PROGRAM Alias
VAR
	i : INT := 1; //mag driver index
	n : INT := 6; //mag driver num
	j : INT := 1; //1-2
	m : INT := 2; //# of ultra cap per driver rack
	k : INT := 1; //ultra cap number 
	
	p : INT := 12; //# of ultra caps = 12
END_VAR

//R1 : MCP**  
	//INPUT
	//AI - EL3068
	MCP_IO.MagDriver[1].ShotCurrentFeedback_raw	:= Input.R1_01_00; //
	MCP_IO.MagDriver[2].ShotCurrentFeedback_raw	:= Input.R1_01_01; //
	MCP_IO.MagDriver[3].ShotCurrentFeedback_raw	:= Input.R1_01_02; // 
	MCP_IO.MagDriver[4].ShotCurrentFeedback_raw	:= Input.R1_01_03; //
	MCP_IO.MagDriver[5].ShotCurrentFeedback_raw	:= Input.R1_01_04; // 
	MCP_IO.MagDriver[6].ShotCurrentFeedback_raw	:= Input.R1_01_05; //  
	//Spare										:= Input.R1_01_06; //  
	//Spare										:= Input.R1_01_07; //
	
	//DI
	MCP_IO.MagDriver[1].DumpResistorTemp_raw	:= Input.R1_02_00; //
	MCP_IO.MagDriver[2].DumpResistorTemp_raw	:= Input.R1_02_01; // 
	MCP_IO.MagDriver[3].DumpResistorTemp_raw	:= Input.R1_02_02; // 
	MCP_IO.MagDriver[4].DumpResistorTemp_raw	:= Input.R1_02_03; // 
	MCP_IO.MagDriver[5].DumpResistorTemp_raw	:= Input.R1_02_04; // 
	MCP_IO.MagDriver[6].DumpResistorTemp_raw	:= Input.R1_02_05; // 
	
	MCP_IO.MagDriver[1].SCR_ready_to_fire		:= Input.R1_03_00; // 
	MCP_IO.MagDriver[2].SCR_ready_to_fire		:= Input.R1_03_01; // 
	MCP_IO.MagDriver[3].SCR_ready_to_fire		:= Input.R1_03_02; // 
	MCP_IO.MagDriver[4].SCR_ready_to_fire		:= Input.R1_03_03; // 
	MCP_IO.MagDriver[5].SCR_ready_to_fire		:= Input.R1_03_04; // 
	MCP_IO.MagDriver[6].SCR_ready_to_fire		:= Input.R1_03_05; // 
	
	MCP_IO.MagDriver[1].ChargeRelayClose		:= Input.R1_04_00; //
	MCP_IO.MagDriver[2].ChargeRelayClose		:= Input.R1_04_01; //
	MCP_IO.MagDriver[3].ChargeRelayClose		:= Input.R1_04_02; //
	MCP_IO.MagDriver[4].ChargeRelayClose		:= Input.R1_04_03; //
	MCP_IO.MagDriver[5].ChargeRelayClose		:= Input.R1_04_04; //
	MCP_IO.MagDriver[6].ChargeRelayClose		:= Input.R1_04_05; //
	
	//DQ
	Output.R1_05_00	:= MCP_IO.MagDriver[1].CloseChargeRly;
	Output.R1_05_01	:= MCP_IO.MagDriver[2].CloseChargeRly;
	Output.R1_05_02	:= MCP_IO.MagDriver[3].CloseChargeRly;
	Output.R1_05_03	:= MCP_IO.MagDriver[4].CloseChargeRly;
	Output.R1_05_04	:= MCP_IO.MagDriver[5].CloseChargeRly;
	Output.R1_05_05	:= MCP_IO.MagDriver[6].CloseChargeRly;
	//Output.R1_05_06	:= 
	//Output.R1_05_07	:= 
	
	//DQ
	Output.R1_06_00	:= MCP_IO.MagDriver[1].OpenDumpRly;
	Output.R1_06_01	:= MCP_IO.MagDriver[2].OpenDumpRly;
	Output.R1_06_02	:= MCP_IO.MagDriver[3].OpenDumpRly;
	Output.R1_06_03	:= MCP_IO.MagDriver[4].OpenDumpRly;
	Output.R1_06_04 := MCP_IO.MagDriver[5].OpenDumpRly;
	Output.R1_06_05 := MCP_IO.MagDriver[6].OpenDumpRly;
	Output.R1_06_06 := MCP_IO.TriggerScope;
	
	MCP_IO.MagDriver[1].DumpRelayOpen		:= Input.R1_07_00; //
	MCP_IO.MagDriver[2].DumpRelayOpen		:= Input.R1_07_01; //
	MCP_IO.MagDriver[3].DumpRelayOpen		:= Input.R1_07_02; //
	MCP_IO.MagDriver[4].DumpRelayOpen		:= Input.R1_07_03; //
	MCP_IO.MagDriver[5].DumpRelayOpen		:= Input.R1_07_04; //
	MCP_IO.MagDriver[6].DumpRelayOpen		:= Input.R1_07_05; //
	(*shaft ramp add below*)
	
	//DQ
	Output.R1_08_00	:= MCP_IO.Charger[1].inhibit;
	Output.R1_08_01	:= MCP_IO.Charger[2].inhibit;
	Output.R1_08_02	:= MCP_IO.Charger[3].inhibit;
	Output.R1_08_03	:= MCP_IO.Charger[4].inhibit;
	Output.R1_08_04	:= MCP_IO.Charger[5].inhibit;
	Output.R1_08_05	:= MCP_IO.Charger[6].inhibit;
	Output.R1_08_06 := MCP_IO.TriggerSCRs;
	Output.R1_08_07	:= MCP_IO.TurnONSystemChargedLED;
		
	//EL4008 AQ
	Output.R1_09_00	:= MCP_IO.Charger[1].voltageSP_raw;
	Output.R1_09_01	:= MCP_IO.Charger[2].voltageSP_raw;
	Output.R1_09_02	:= MCP_IO.Charger[3].voltageSP_raw;
	Output.R1_09_03	:= MCP_IO.Charger[4].voltageSP_raw;	
	Output.R1_09_04	:= MCP_IO.Charger[5].voltageSP_raw;
	Output.R1_09_05	:= MCP_IO.Charger[6].voltageSP_raw;
	
	//CANBUS 
	//Output.R1_10_CANrequest := CAN_comm.
	Output.R1_10_CANrequest.cobId := MCP_IO.MagDriver[1].Cap[1].CanTx_config_ID;
	Output.R1_10_CANrequest.data[0] := MCP_IO.MagDriver[1].Cap[1].CanTx_config_request[0];
	Output.R1_10_CANrequest.data[1] := MCP_IO.MagDriver[1].Cap[1].CanTx_config_request[1];
	Output.R1_10_CANrequest.data[2] := MCP_IO.MagDriver[1].Cap[1].CanTx_config_request[2];
	Output.R1_10_CANrequest.data[3] := MCP_IO.MagDriver[1].Cap[1].CanTx_config_request[3];
	Output.R1_10_CANrequest.data[4] := MCP_IO.MagDriver[1].Cap[1].CanTx_config_request[4];
	Output.R1_10_CANrequest.data[5] := MCP_IO.MagDriver[1].Cap[1].CanTx_config_request[5];
	Output.R1_10_CANrequest.data[6] := MCP_IO.MagDriver[1].Cap[1].CanTx_config_request[6];
	Output.R1_10_CANrequest.data[7] := MCP_IO.MagDriver[1].Cap[1].CanTx_config_request[7];
	
	// P1 PP comm
	HMI_DB.ClearFaultPB := plc_plc_comm_DB.Button.ClearAllFaults;
	HMI_DB.FirePB 		:= plc_plc_comm_DB.Button.FirePBPressed;
	HMI_DB.DumpPB 		:= plc_plc_comm_DB.Button.DumpPB;

	//MCP_IO.MagDriver[1].Cap[1].Elec_AveVolt 		:= Input.R1_10_CapNumber[1].Status.Elec_AveVolt; //per cell <- example
	//this is replaced by the loop below
(*	MCP_IO.MagDriver[1].Cap[1].Elec_AveVolt 		:= Input.R1_10_CapNumber[1].Status.Elec_AveVolt; //per cell
	MCP_IO.MagDriver[1].Cap[1].Elec_Balancing 		:= Input.R1_10_CapNumber[1].Status.Elec_Balancing; // 0x0[Not Active], 0x1[Active], 0x2[Error], 0x3[Not Available]
	MCP_IO.MagDriver[1].Cap[1].Elec_HighestVolt 	:= Input.R1_10_CapNumber[1].Status.Elec_HighestVolt; //per cell
	MCP_IO.MagDriver[1].Cap[1].Elec_Imbalance 		:= Input.R1_10_CapNumber[1].Status.Elec_Imbalance;  // 0x0[No Warnings], 0x1[Warning Active], 0x2[Alarm Active], 0x3[Not Available]
	MCP_IO.MagDriver[1].Cap[1].Elec_OverVoltage		:= Input.R1_10_CapNumber[1].Status.Elec_OverVoltage;  // 0x0[No Warnings], 0x1[Warning Active], 0x2[Alarm Active], 0x3[NOT Available] 
	MCP_IO.MagDriver[1].Cap[1].Elec_VoltageSum		:= Input.R1_10_CapNumber[1].Status.Elec_VoltageSum; //total voltage in one UC
	MCP_IO.MagDriver[1].Cap[1].Therm_HighestCell	:= Input.R1_10_CapNumber[1].Status.Therm_HighestCell; //C
	MCP_IO.MagDriver[1].Cap[1].Therm_HighTemp		:= Input.R1_10_CapNumber[1].Status.Therm_HighTemp;  //0x0[No Warnings], 0x1[Warning Active], 0x2[Alarm Active], 0x3[NOT Available]
*)	
//need to verify the couunter
	FOR i := 1 TO n BY 1 DO 
		FOR j := 1 TO m BY 1 DO 
			IF j = 1 THEN 
				k := 2*i -j;
				ELSIF j = 2 THEN 
					k :=j*i;
			END_IF

			MCP_IO.MagDriver[i].Cap[j].Elec_AveVolt			:= Input.R1_10_CapNumber[k].Elec_AveVolt; //per cell
			MCP_IO.MagDriver[i].Cap[j].Elec_Balancing		:= Input.R1_10_CapNumber[k].Elec_Balancing; // 0x0[Not Active], 0x1[Active], 0x2[Error], 0x3[Not Available]
			MCP_IO.MagDriver[i].Cap[j].Elec_HighestVolt		:= Input.R1_10_CapNumber[k].Elec_HighestVolt; //per cell
			MCP_IO.MagDriver[i].Cap[j].Elec_Imbalance		:= Input.R1_10_CapNumber[k].Elec_Imbalance;  // 0x0[No Warnings], 0x1[Warning Active], 0x2[Alarm Active], 0x3[Not Available]
			MCP_IO.MagDriver[i].Cap[j].Elec_OverVoltage		:= Input.R1_10_CapNumber[k].Elec_OverVoltage;  // 0x0[No Warnings], 0x1[Warning Active], 0x2[Alarm Active], 0x3[NOT Available] 
			MCP_IO.MagDriver[i].Cap[j].Elec_VoltageSum		:= Input.R1_10_CapNumber[k].Elec_VoltageSum; //total voltage in one UC
			MCP_IO.MagDriver[i].Cap[j].Therm_HighestCell	:= Input.R1_10_CapNumber[k].Therm_HighestCell; //C
			MCP_IO.MagDriver[i].Cap[j].Therm_HighTemp		:= Input.R1_10_CapNumber[k].Therm_HighTemp;  //0x0[No Warnings], 0x1[Warning Active], 0x2[Alarm Active], 0x3[NOT Available]

		END_FOR		
	END_FOR
	
	MCP_IO.MagDriver[1].Cap[1].UltraCap_Dummy.R1_10_UC_Rx_cobID := Input.R1_10_UC_7F_status.R1_10_UC_Rx_cobID;
	MCP_IO.MagDriver[1].Cap[1].UltraCap_Dummy.R1_10_UC_Rx_data := Input.R1_10_UC_7F_status.R1_10_UC_Rx_data;	
	// need to have how many voltage monitor board or voltage transmitter board per fruit stand ????
	//LCP3_IO.VMB.VTB[1].

	//LV Alias
	//commented out to test the sequence
	(*
	HMI_DB.ChargePB 				:= LV.TxWord1.0;
	HMI_DB.DumpPB					:= LV.TxWord1.1;		
	HMI_DB.AbortPB					:= LV.TxWord1.2;
	HMI_DB.FirePB					:= LV.TxWord1.3;
	HMI_DB.ClearFaultPB 			:= LV.TxWord1.4;
	HMI_DB.AllDumpRelaysOpenBP		:= LV.TxWord1.5;
	HMI_DB.AllChargeRelayCloseBP	:= LV.TxWord1.6;
	HMI_DB.SystemSafeBP				:= LV.TxWord1.7;
	HMI_DB.CloseChargeRlySW			:= LV.TxWord1.8;
	HMI_DB.OpenDumpRlySW 			:= LV.TxWord1.9;
	HMI_DB.HMI_ManualModeSelected	:= LV.TxWord1.10;  // 1 = manual mode selected
	HMI_DB.TurnChrgHVonSW			:= LV.TxWord1.11;
	HMI_DB.TurnChrgInhibitOffSW		:= LV.TxWord1.12;
	HMI_DB.TurnOnShotTrigSW			:= LV.TxWord1.13;
	HMI_DB.TurnOnChargeAlarm		:= LV.TxWord1.14;
	HMI_DB.AllVoltMonBoardStatusOKBP:= LV.TxWord1.15;
	//not sure if you want to control these via LV
	(*
	MCP_IO.Charger[1].HV_ON			:= LV.TxWord2.0;
	MCP_IO.Charger[1].inhibit		:= LV.TxWord2.1;
	MCP_IO.Charger[2].HV_ON			:= LV.TxWord2.2;
	MCP_IO.Charger[2].inhibit		:= LV.TxWord2.3;
	
	MCP_IO.Charger[3].HV_ON			:= LV.TxWord2.4;
	MCP_IO.Charger[3].inhibit		:= LV.TxWord2.5;
	MCP_IO.Charger[4].HV_ON			:= LV.TxWord2.6;
	MCP_IO.Charger[4].inhibit		:= LV.TxWord2.7;
	MCP_IO.Charger[5].HV_ON			:= LV.TxWord2.8;
	MCP_IO.Charger[5].inhibit		:= LV.TxWord2.9;
	MCP_IO.Charger[6].HV_ON			:= LV.TxWord2.10;
	MCP_IO.Charger[6].inhibit		:= LV.TxWord2.11;
	HMI_DB.HMI_DB.AllDumpRelaysCloseBP := LV.TxWord2.12;
	*)
	
	LV.RxWord1.0 := LV.Charger[1].EndOfCharge			:= MCP_IO.Charger[1].EndOfCharge;
	LV.RxWord1.1 := LV.Charger[1].HV_isON				:= MCP_IO.Charger[1].HV_isON;
	LV.RxWord1.2 := LV.Charger[1].inhibited				:= MCP_IO.Charger[1].inhibited;
	LV.RxWord1.3 := LV.Charger[1].SummaryFaulted		:= MCP_IO.Charger[1].SummaryFaulted;
	LV.RxWord1.4 := LV.Charger[2].EndOfCharge			:= MCP_IO.Charger[2].EndOfCharge;
	LV.RxWord1.5 := LV.Charger[2].HV_isON				:= MCP_IO.Charger[2].HV_isON;
	LV.RxWord1.6 := LV.Charger[2].inhibited				:= MCP_IO.Charger[2].inhibited;
	LV.RxWord1.7 := LV.Charger[2].SummaryFaulted		:= MCP_IO.Charger[2].SummaryFaulted;
	LV.RxWord1.8 := LV.Charger[3].EndOfCharge			:= MCP_IO.Charger[3].EndOfCharge;
	LV.RxWord1.9 := LV.Charger[3].HV_isON				:= MCP_IO.Charger[3].HV_isON;
	LV.RxWord1.10 := LV.Charger[3].inhibited			:= MCP_IO.Charger[3].inhibited;
	LV.RxWord1.11 := LV.Charger[3].SummaryFaulted		:= MCP_IO.Charger[3].SummaryFaulted;
	LV.RxWord1.12 := LV.Charger[4].EndOfCharge			:= MCP_IO.Charger[4].EndOfCharge;
	LV.RxWord1.13 := LV.Charger[4].HV_isON				:= MCP_IO.Charger[4].HV_isON;
	LV.RxWord1.14 := LV.Charger[4].inhibited			:= MCP_IO.Charger[4].inhibited;
	LV.RxWord1.15 := LV.Charger[4].SummaryFaulted		:= MCP_IO.Charger[4].SummaryFaulted;
	
	LV.RxWord2.0 := LV.Charger[5].EndOfCharge			:= MCP_IO.Charger[5].EndOfCharge;
	LV.RxWord2.1 := LV.Charger[5].HV_isON				:= MCP_IO.Charger[5].HV_isON;
	LV.RxWord2.2 := LV.Charger[5].inhibited				:= MCP_IO.Charger[5].inhibited;
	LV.RxWord2.3 := LV.Charger[5].SummaryFaulted		:= MCP_IO.Charger[5].SummaryFaulted;
	LV.RxWord2.4 := LV.Charger[6].EndOfCharge			:= MCP_IO.Charger[6].EndOfCharge;
	LV.RxWord2.5 := LV.Charger[6].HV_isON				:= MCP_IO.Charger[6].HV_isON;
	LV.RxWord2.6 := LV.Charger[6].inhibited				:= MCP_IO.Charger[6].inhibited;
	LV.RxWord2.7 := LV.Charger[6].SummaryFaulted		:= MCP_IO.Charger[6].SummaryFaulted;
	(*shaft ramp add below*)
	
	LV.RxWord3.0 := LCP1_IO.Segment[1].ChargeRly_close;
	LV.RxWord3.1 := LCP1_IO.Segment[2].ChargeRly_close;
	LV.RxWord3.2 := LCP1_IO.Segment[3].ChargeRly_close;
	LV.RxWord3.3 := LCP2_IO.Segment[4].ChargeRly_close;
	LV.RxWord3.4 := LCP2_IO.Segment[5].ChargeRly_close;
	LV.RxWord3.5 := LCP2_IO.Segment[6].ChargeRly_close;
	
	LV.RxWord3.6 := LCP1_IO.Segment[1].Module1To3DumpRly_close;
	LV.RxWord3.7 := LCP1_IO.Segment[2].Module4To6DumpRly_close;
	LV.RxWord3.8 := LCP1_IO.Segment[3].Module7To9DumpRly_close;
	LV.RxWord3.9 := LCP2_IO.Segment[4].Module1To3DumpRly_close;
	LV.RxWord3.10 := LCP2_IO.Segment[5].Module4To6DumpRly_close;
	LV.RxWord3.11 := LCP2_IO.Segment[6].Module7To9DumpRly_close; 
	//LV.RxWord3.12  
	//LV.RxWord3.13  
	//LV.RxWord3.14  
	//LV.RxWord3.15  
	
	HMI_DB.ChargerHVOFF_rlyDelayPT_INT	:= LV.TxInt[1];
	HMI_DB.HVONdelayPT_INT 				:= LV.TxInt[2];
	LV.RxInt[1]							:= HMI_DB.ChargingRunOutTMR_elapse;
	
	HMI_DB.RunOutTMR_PT_INT				:= LV.TxDint[1];
	LV.RxDint[1]						:= HMI_DB.RunOutTMR_elapse;	
	
	
	FOR i := 1 TO n BY 1 DO
		HMI_DB.TDKLoad[i].eChargerType 					:= LV.TDKLoad[i].eChargerType;
		HMI_DB.TDKLoad[i].PSratedV						:= LV.TDKLoad[i].PSratedV;
		HMI_DB.TDKLoad[i].RequiredChargedV 				:= LV.TDKLoad[i].RequiredChargedV;
		HMI_DB.TDKLoad[i].wLCA							:= LV.TDKLoad[i].wLCA;;
		HMI_DB.TDKLoad[i].NumOfCharger					:= LV.TDKLoad[i].NumOfCharger;	
		HMI_DB.TDKLoad[i].TotalCapacitance				:= LV.TDKLoad[i].TotalCapacitance;

		LV.Charger[i].ChargeTime 						:= MCP_IO.Charger[i].ChargeTime;
		LV.RxREAL[i] := LV.Charger[i].voltageFeedback	:= MCP_IO.Charger[i].voltageFeedback; //LV.RxREAL[8] for shaft ramp
		MCP_IO.Charger[i].voltageSP (*make this real*)	:= LV.TxREAL[i] := LV.Charger[i].voltageSP;
	
	END_FOR
	
	 //lcp 1 cap volt to lv
		 LV.RxREAL[9] := LCP1_IO.Segment[1].Module[1].VoltageFeedback[1];
		 LV.RxREAL[10] := LCP1_IO.Segment[1].Module[1].VoltageFeedback[2];
		 LV.RxREAL[11] := LCP1_IO.Segment[1].Module[2].VoltageFeedback[1];
		 LV.RxREAL[12] := LCP1_IO.Segment[1].Module[2].VoltageFeedback[2];
		 LV.RxREAL[13] := LCP1_IO.Segment[1].Module[3].VoltageFeedback[1];
		 LV.RxREAL[14] := LCP1_IO.Segment[1].Module[3].VoltageFeedback[2];
		 
		 LV.RxREAL[15] := LCP1_IO.Segment[2].Module[4].VoltageFeedback[1];
		 LV.RxREAL[16] := LCP1_IO.Segment[2].Module[4].VoltageFeedback[2];
		 LV.RxREAL[17] := LCP1_IO.Segment[2].Module[5].VoltageFeedback[1];
		 LV.RxREAL[18] := LCP1_IO.Segment[2].Module[5].VoltageFeedback[2];
		 LV.RxREAL[19] := LCP1_IO.Segment[2].Module[6].VoltageFeedback[1];
		 LV.RxREAL[20] := LCP1_IO.Segment[2].Module[6].VoltageFeedback[2];
		 
		 LV.RxREAL[21] := LCP1_IO.Segment[3].Module[7].VoltageFeedback[1];
		 LV.RxREAL[22] := LCP1_IO.Segment[3].Module[7].VoltageFeedback[2];
		 LV.RxREAL[23] := LCP1_IO.Segment[3].Module[8].VoltageFeedback[1];
		 LV.RxREAL[24] := LCP1_IO.Segment[3].Module[8].VoltageFeedback[2];
		 LV.RxREAL[25] := LCP1_IO.Segment[3].Module[9].VoltageFeedback[1];
		 LV.RxREAL[26] := LCP1_IO.Segment[3].Module[9].VoltageFeedback[2];
		 
	//lcp2 cap volt to lv	 
		 LV.RxREAL[27] := LCP2_IO.Segment[4].Module[1].VoltageFeedback[1];
		 LV.RxREAL[28] := LCP2_IO.Segment[4].Module[1].VoltageFeedback[2];
		 LV.RxREAL[29] := LCP2_IO.Segment[4].Module[2].VoltageFeedback[1];
		 LV.RxREAL[30] := LCP2_IO.Segment[4].Module[2].VoltageFeedback[2];
		 LV.RxREAL[31] := LCP2_IO.Segment[4].Module[3].VoltageFeedback[1];
		 LV.RxREAL[32] := LCP2_IO.Segment[4].Module[3].VoltageFeedback[2];
		
		 LV.RxREAL[33] := LCP2_IO.Segment[5].Module[4].VoltageFeedback[1];
		 LV.RxREAL[34] := LCP2_IO.Segment[5].Module[4].VoltageFeedback[2];
		 LV.RxREAL[35] := LCP2_IO.Segment[5].Module[5].VoltageFeedback[1];
		 LV.RxREAL[36] := LCP2_IO.Segment[5].Module[5].VoltageFeedback[2];
		 LV.RxREAL[37] := LCP2_IO.Segment[5].Module[6].VoltageFeedback[1];
		 LV.RxREAL[38] := LCP2_IO.Segment[5].Module[6].VoltageFeedback[2];
		 
		 LV.RxREAL[39] := LCP2_IO.Segment[6].Module[7].VoltageFeedback[1];
		 LV.RxREAL[40] := LCP2_IO.Segment[6].Module[7].VoltageFeedback[2];
		 LV.RxREAL[41] := LCP2_IO.Segment[6].Module[8].VoltageFeedback[1];
		 LV.RxREAL[42] := LCP2_IO.Segment[6].Module[8].VoltageFeedback[2];
		 LV.RxREAL[43] := LCP2_IO.Segment[6].Module[9].VoltageFeedback[1];
		 LV.RxREAL[44] := LCP2_IO.Segment[6].Module[9].VoltageFeedback[2];
		 *)
	

IF j > m THEN 
	j := 1;
END_IF

IF i > n THEN 
	i := 1;
END_IF

IF k > p THEN 
	k := 1;
END_IF

END_PROGRAM

(* stored: Version 1.1.0.1, ProductVersion 3.1.4024.11
   POU Alias: Id {ebc75665-f0df-4b03-b4d1-48515468f179}, SpecialFunc None *)
